{attribute 'qualified_only'}
{attribute 'strict'}
TYPE E_CPUType :
(
    CX5130 := 0,
    C6017_0020 := 1
);
END_TYPE

(* stored: Version 1.1.0.1, ProductVersion 3.1.4024.11
   DUT E_CPUType: Id {78ea3fa6-b103-4c1f-b5a7-d343f24fda9f} *)
